PROGRAM MAIN
VAR	
	{attribute wpf [Container(Layout.Stack)]}	
	{attribute addProperty Name "WPF cyclinder"}
	_wpfCyclinder : fbCylinder;	
	{attribute wpf [Container(Layout.Stack)]}	
	{attribute addProperty Name "WPF cyclinder 1"}
	_wpfCyclinder_1 : fbCylinder;
	{attribute wpf [Container(Layout.Stack)]}	
	{attribute addProperty Name "WPF cyclinder 2"}
	_wpfCyclinder_2 : fbCylinder;
	{attribute wpf [Container(Layout.Stack)]}	
	{attribute addProperty Name "WPF cyclinder 3"}
	_wpfCyclinder_3 : fbCylinder;	
END_VAR

_wpfCyclinder(inAtHomePos:=IO.A1[0] , inAtWorkPos:=IO.A1[1] , outToHomePos=> IO.A2[0], outToWorkPos=>IO.A2[1]);

_wpfCyclinder.Manual();
_wpfCyclinder_1.Manual();
_wpfCyclinder_2.Manual();
_wpfCyclinder_3.Manual();

END_PROGRAM

(* stored: Version 1.1.0.1, ProductVersion 3.1.4024.5
   POU MAIN: Id {f20f72a3-44bd-4b01-bab9-6aeb1376a30d}, SpecialFunc None *)
